FUNCTION_BLOCK CL_AxisDriverAX8206 EXTENDS CL_CardCom
VAR
  bInit                   : BOOL := FALSE;
  _stDriverCom_P          : POINTER TO ST_DriverAX8206_HWI;
  _stDriverCh_P           : POINTER TO ST_ChannelAX8206_HWI;
END_VAR

IF bInit THEN
  THIS^.Run();
END_IF

METHOD PROTECTED InitDefect : BOOL
VAR_INPUT
END_VAR
InitDefect := true;
END_METHOD

METHOD PUBLIC InitDriver : BOOL
VAR_INPUT
  stDriverCom_P     : POINTER TO ST_DriverAX8206_HWI;
  stDriverCh_P      : POINTER TO ST_ChannelAX8206_HWI;
END_VAR
InitDriver := FALSE;
IF stDriverCom_P <> 0 AND stDriverCh_P <> 0 AND NOT bInit THEN
  _stDriverCom_P := stDriverCom_P;
  _stDriverCh_P := stDriverCh_P;
  bInit := InitDriver := InitCom(stCardStateIn_P := ADR(_stDriverCom_P^.comState)) AND  InitDefect() AND InitDefectCom();
END_IF
END_METHOD

METHOD PRIVATE Run
VAR_INPUT
END_VAR
END_METHOD

END_FUNCTION_BLOCK

(* stored: Version 1.1.0.1, ProductVersion 3.1.4024.12
   POU CL_AxisDriverAX8206: Id {c28f2ae3-7ac4-4e6e-83ad-c702b6dc71e8}, SpecialFunc None
   Method InitDefect: Id {73fa3589-ebd6-4c1f-92bb-37f72a7474db}
   Method InitDriver: Id {bb8bf61f-ae7c-41ad-9f90-fcbffd12ec34}
   Method Run: Id {1277389a-916b-454f-ab5b-820e51c371c2} *)
